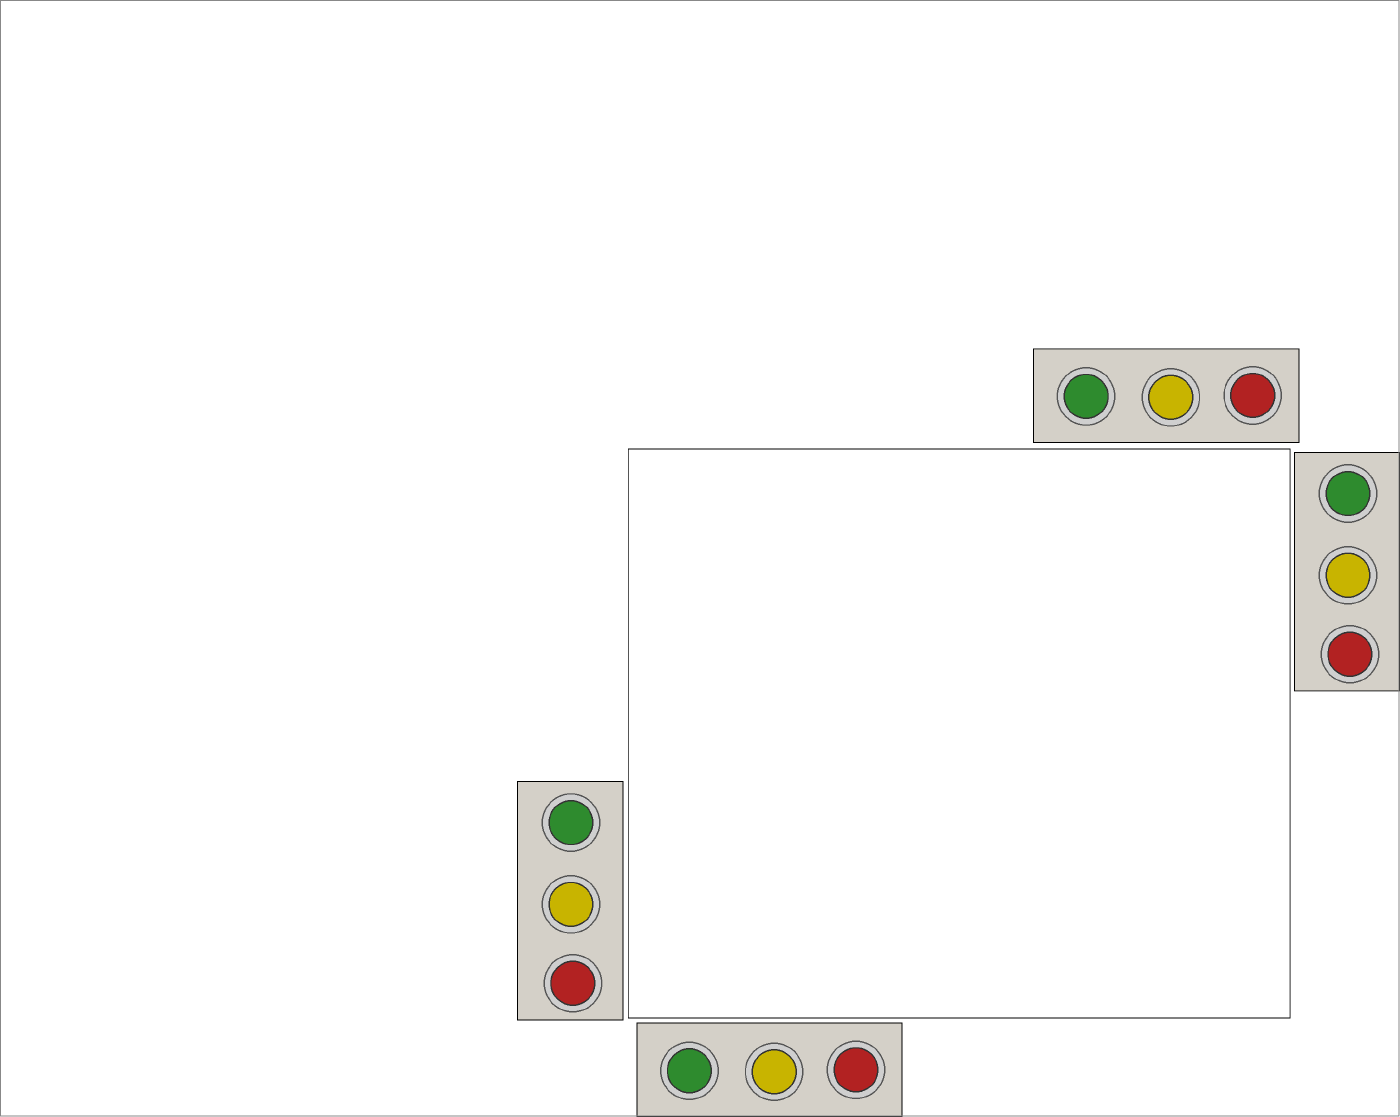
VISUALIZATION Visualization  // 1454x1161
    Group (1073,362 276x98)
        Rectangle (0,0 276x98)
        Lamp1 (20,15 70x70), variable: TrafficLgiht.bNorthGreenLight, style: Lamp-Lamp1-Green
        Lamp1 (193,14 70x70), variable: TrafficLgiht.bNorthRedLight, style: Lamp-Lamp1-Red
        Lamp1 (108,16 70x70), variable: TrafficLgiht.bNorthYellowLight, style: Lamp-Lamp1-Yellow
    Group (537,812 110x248)
        Rectangle (0,0 110x248)
        Lamp1 (21,8 70x70), variable: TrafficLgiht.bWestGreenLight, style: Lamp-Lamp1-Green
        Lamp1 (23,175 70x70), variable: TrafficLgiht.bWestRedLight, style: Lamp-Lamp1-Red
        Lamp1 (21,93 70x70), variable: TrafficLgiht.bWestYellowLight, style: Lamp-Lamp1-Yellow
    Rectangle (652,466 688x592)
    Group (661,1063 276x98)
        Rectangle (0,0 276x98)
        Lamp1 (20,15 70x70), variable: TrafficLgiht.bNorthGreenLight, style: Lamp-Lamp1-Green
        Lamp1 (193,14 70x70), variable: TrafficLgiht.bNorthRedLight, style: Lamp-Lamp1-Red
        Lamp1 (108,16 70x70), variable: TrafficLgiht.bNorthYellowLight, style: Lamp-Lamp1-Yellow
    Group (1344,470 110x248)
        Rectangle (0,0 110x248)
        Lamp1 (21,8 70x70), variable: TrafficLgiht.bWestGreenLight, style: Lamp-Lamp1-Green
        Lamp1 (23,175 70x70), variable: TrafficLgiht.bWestRedLight, style: Lamp-Lamp1-Red
        Lamp1 (21,93 70x70), variable: TrafficLgiht.bWestYellowLight, style: Lamp-Lamp1-Yellow
END_VISUALIZATION

(* stored: Version 1.1.0.1, ProductVersion 3.1.4024.11
   Visu Visualization: Id {89bb90e2-9c1d-4ce2-a69d-bca2bc910bfb} *)
